PROGRAM MAIN
VAR
	counter : INT := 0;
	
	Setup : BOOL := TRUE;
	
	// AI Scaling to percent
	AI_Low : INT := 3375; 
	AI_High : INT := 20200;
	AI0_scaled : INT := 0;
	
	// led toggle rates (Hz)
	toggleRate : INT := 1;
	toggleRateMax : INT := 100;
	toggleRateMin : INT := 1;
	toggleEnable: BOOL := FALSE;
END_VAR

// setup
IF Setup THEN
	GVL.DO0 := FALSE;
	GVL.DO1 := TRUE;
	
	// setup finished
	Setup := FALSE;
END_IF


// main loop
counter := counter + 100;
IF counter > 30000 THEN
	counter := 0;
END_IF

// scale AI value to percent
AI0_scaled := Scale(GVL.AI0, 
					AI_High, AI_Low,
					toggleRateMax, toggleRateMin);
					
IF GVL.DI0 OR GVL.DI0_OR THEN
	toggleEnable := TRUE;
END_IF

IF GVL.DI1 OR GVL.DI1_OR THEN
	toggleEnable := FALSE;
END_IF

IF toggleEnable THEN
	IF counter > GVL.AI0 THEN
		GVL.DO0 := NOT GVL.DO0;
		GVL.DO1 := NOT GVL.DO1;
		counter := 0;
	END_IF
END_IF

END_PROGRAM

(* stored: Version 1.1.0.1, ProductVersion 3.1.4024.12
   POU MAIN: Id {b3ecad9f-d573-47a2-b344-f69e047572b9}, SpecialFunc None *)
